(* Logix 5000 project; controller R5_CSS vendor 1 type 14 code 74 rev 19.11; software revision 19.01; part 4 of 20 *)
(* tags used below, declared in another part *)
   AlarmMaster : DINT;
   Coal_Tank_Heel_Inches : REAL;
   FC101 : FLOW_CONTROL;   // QUENCH BASIN FLOW TRANSMITTER CONTROL
   FC108 : FLOW_CONTROL;   // QUENCH FEED FLOW TRANSMITTER
   FC140A : FLOW_CONTROL;   // QUENCH TOWER UPPER SPRAY FLOW CONTROL
   FC140B : FLOW_CONTROL;   // QUENCH TOWER LOWER SPRAY FLOW CONTROL
   FC403 : FLOW_CONTROL;   // COALESCER FLOW CONTROLLER FEEDS TCV108
   FCV410_LT_Hold : BOOL;
   FlowControlForce : BOOL;
   FlowControlForceONS : BOOL;
   FT101_SCP : SCLP;   // QUENCH BASIN FLOW TRANSMITTER SCALER
   FT108_SCP : SCLP;   // QUENCH FEED FLOW TRANSMITTER SCALER
   FT140A_SCP : SCLP;   // QUENCH TOWER UPPER SPRAY FIT SCALER
   FT140ABFlowMeterFailed : BOOL;
   FT140B_SCP : SCLP;   // QUENCH TOWER LOWER SPRAY FLOW TRANSMITTER SCALER
   FT403_SCP : SCLP;   // QUENCH CONDITIONING QUENCH WATER PHASE FLOW SCALER
   LC101 : LEVEL_CONTROL;   // QUENCH TOWER BASIN LIT
   LC101_LT_Temp : REAL;
   LC304 : LEVEL_CONTROL;   // SETTLER SECONDARY TANK INTERFACE LEVEL
   LC304_LT_Raw : REAL;
   LevelControlForce : BOOL;
   LevelControlForceONS : BOOL;
   LossOfSignal_mA : DINT;
   LT101_SCP : SCLP;   // QUENCH TOWER BASIN LIT SCALER
   LT304_SCP : SCLP;   // QUENCH COALESCING SEPARATOR SECONDARY CHAMBER LEVEL SCALER
   PC132 : PRESSURE_CONTROL;
   PC132_SCP : SCLP;
   PC133 : PRESSURE_CONTROL;
   PC133_SCP : SCLP;
   PC134 : PRESSURE_CONTROL;
   PC134_SCP : SCLP;
   PC408 : PRESSURE_CONTROL;
   PDT408_SCP : SCLP;
   QuenchFlowAutoControl : BOOL;
   QuenchFlowAutoControlPB : BOOL;
   QuenchFlowAutoControlPB_ONS : BOOL;
   QuenchFlowMeterFailed : BOOL;
   QuenchFlowMeterFailedTOF : TIMER;
   TC101A : TEMP_CONTROL;   // QUENCH BASIN TRANSFER BASIN A TEMPERATURE CONTROL
   TC101B : TEMP_CONTROL;   // QUENCH BASIN TRANSFER BASIN B TEMPERATURE CONTROL
   TC110 : TEMP_CONTROL;   // Quench Water Cartridge Heater Bundle Temp
   TC110_SCP : SCLP;
   TC112 : TEMP_CONTROL;   // Quench Water Cartridge Heater ProcessTemp
   TC112_SCP : SCLP;
   TC114A : TEMP_CONTROL;   // QUENCH BASIN SHELL TEMPERATURE CONTROL
   TC114B : TEMP_CONTROL;   // QUENCH BASIN LIQUID TEMPERATURE CONTROL
   TC121C : TEMP_CONTROL;   // GTL FROM PRUC TEMPERATURE CONTROL
   TC121D : TEMP_CONTROL;   // GTL FROM PRUD TEMPERATURE CONTROL
   TC121E : TEMP_CONTROL;
   TC121F : TEMP_CONTROL;
   TC121G : TEMP_CONTROL;
   TC121H : TEMP_CONTROL;
   TC123A : TEMP_CONTROL;   // HEAT JACKET VENT FROM PRUA TEMPERATURE CONTROL
   TC123A_SCP : SCLP;   // HEAT JACKET VENT FROM PRUA TEMPERATURE TRANSMITTER SCALER
   TC123B : TEMP_CONTROL;
   TC123B_SCP : SCLP;   // HEAT JACKET VENT FROM PRUB TEMPERATURE TRANSMITTER SCALER
   TC123C : TEMP_CONTROL;   // HEAT JACKET VENT FROM PRUC TEMPERATURE CONTROL
   TC123C_SCP : SCLP;   // HEAT JACKET VENT FROM PRUC TEMPERATURE TRANSMITTER SCALER
   TC123D : TEMP_CONTROL;   // HEAT JACKET VENT FROM PRUD TEMPERATURE TRANSMITTER
   TC123D_SCP : SCLP;   // HEAT JACKET VENT FROM PRUD TEMPERATURE TRANSMITTER SCALER
   TC123E : TEMP_CONTROL;
   TC123E_SCP : SCLP;
   TC123F : TEMP_CONTROL;
   TC123F_SCP : SCLP;
   TC123G : TEMP_CONTROL;
   TC123G_SCP : SCLP;
   TC123H : TEMP_CONTROL;
   TC123H_SCP : SCLP;
   TC135 : TEMP_CONTROL;
   TC135_SCP : SCLP;
   TC136 : TEMP_CONTROL;
   TC136_SCP : SCLP;
   TC137 : TEMP_CONTROL;
   TC137_SCP : SCLP;
   TC215 : TEMP_CONTROL;   // OVERHEAD CONDENSER CHILLED WATER TEMPERATURE TRANSMITTER CONTROL
   TC215_SCP : SCLP;   // OVERHEAD CONDENSER CHILLED WATER TEMPERATURE TRANSMITTER SCALER
   TC216 : TEMP_CONTROL;   // OVERHEAD CONDENSER BASIN TEMPERATURE CONTROL
   TC217 : TEMP_CONTROL;   // OVERHEAD CONDENSED CHILLED WATER RETURN TEMPERATURE CONTROL
   TC218 : TEMP_CONTROL;   // OVERHEAD CONDENSER CHILLED WATER SUPPLY TEMPERATURE CONTROL
   TC313A : TEMP_CONTROL;   // PRIMARY COALESCER SEPARATOR TEMPERATURE CONTROL
   TC313B : TEMP_CONTROL;   // PRIMARY COALESCER SHELL TEMPERATURE CONTROL
   TC319 : TEMP_CONTROL;   // COALESCER OIL CHAMBER PROCESS TEMPERATURE CONTROL
   TC319A : TEMP_CONTROL;   // COALESCER OIL CHAMBER SHEATH TEMPERATURE
   TC320 : TEMP_CONTROL;   // COALESCER OIL CHAMBER SHELL TEMPERATURE TRANSMITTER CONTROL
   TC321A : TEMP_CONTROL;   // COALESCER OIL CHAMBER TRANSFER PUMP A TEMPERATURE TRANSMITTER
   TC321B : TEMP_CONTROL;   // COALESCER OIL CHAMBER TRANSFER PUMP B TEMPERATURE TRANSMITTER
   TC406 : TEMP_CONTROL;   // PROCESS WATER POST HX TEMPERATURE CONTROL
   TC406_SCP : SCLP;   // PROCESS WATER POST HX TEMPERATURE TRANSMITTER SCALER
   TC409 : TEMP_CONTROL;   // HX COOLING WATER SUPPLY TEMPERATURE CONTROL
   TC409_SCP : SCLP;   // HX COOLING WATER SUPPLY TEMPERATURE TRANSMITTER SCALER
   TC410 : TEMP_CONTROL;   // HX COOLING WATER RETURN TEMPERATURE CONTROL
   TC410_SCP : SCLP;   // HX COOLING WATER RETURN TEMPERATURE TRANSMITTER SCALER
   TT101A_SCP : SCLP;   // QUENCH BASIN TRANSFER BASIN A TEMPERATURE TRANSMITTER SCALER
   TT101B_SCP : SCLP;   // QUENCH BASIN TRANSFER BASIN B TEMPERATURE TRANSMITTER SCALER
   TT114A_SCP : SCLP;   // QUENCH BASIN SHELL TEMPERATURE TRANSMITTER SCALER
   TT114B_SCP : SCLP;   // QUENCH BASIN LIQUID TEMPERATURE TRANSMITTER SCALER
   TT121C_SCP : SCLP;
   TT121D_SCP : SCLP;
   TT121E_SCP : SCLP;
   TT121F_SCP : SCLP;   // GTL FROM PRUB TEMPERATURE TRANSMITTER SCALER
   TT121G_SCP : SCLP;   // GTL FROM PRUC TEMPERATURE TRANSMITTER SCALER
   TT121H_SCP : SCLP;   // GTL FROM PRUD TEMPERATURE TRANSMITTER SCALER
   TT216_SCP : SCLP;   // OVERHEAD CONDENSER BASIN TEMPERATURE TRANSMITTER SCALER
   TT217_SCP : SCLP;   // OVERHEAD CONDENSED CHILLED WATER RETURN TEMPERATURE TRANSMITTER
   TT218_SCP : SCLP;   // OVERHEAD CONDENSER CHILLED WATER SUPPLY TEMPERATURE SCALER
   TT313A_SCP : SCLP;   // PRIMARY COALESCER SEPARATOR TEMPERATURE TRANSMITTER SCALER
   TT313B_SCP : SCLP;   // PRIMARY COALESCER SHELL TEMPERATURE TRANSMITTER SCALER
   TT319_SCP : SCLP;   // COALESCER OIL CHAMBER SHELL TEMPERATURE TRANSMITTER SCALER
   TT319A_SCP : SCLP;
   TT320_SCP : SCLP;   // COALESCER OIL CHAMBER SHELL TEMPERATURE TRANSMITTER SCALER
   TT321A_SCP : SCLP;   // COALESCER OIL CHAMBER TRANSFER PUMP A TEMPERATURE TRANSMITTER SCALER
   TT321B_SCP : SCLP;   // COALESCER OIL CHAMBER TRANSFER PUMP B TEMPERATURE TRANSMITTER
(* MainProgram, continued *)

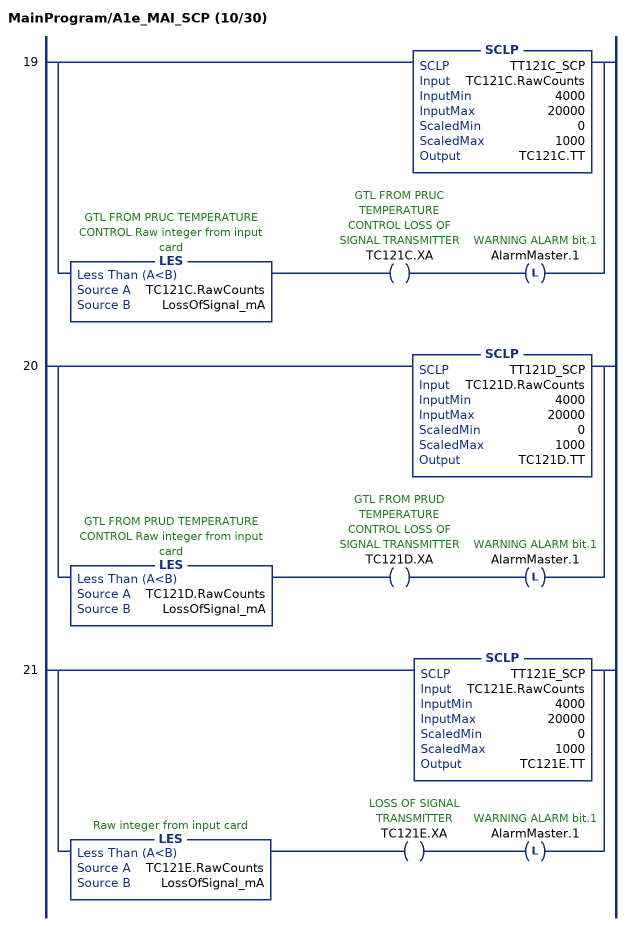
   [picture p54: MainProgram/A1e_MAI_SCP rungs 19-21]
   19: [SCLP(TT121C_SCP,TC121C.RawCounts,4000,20000,0,1000,TC121C.TT) ,LES(TC121C.RawCounts,LossOfSignal_mA) OTE(TC121C.XA) OTL(AlarmMaster.1) ];
   20: [SCLP(TT121D_SCP,TC121D.RawCounts,4000,20000,0,1000,TC121D.TT) ,LES(TC121D.RawCounts,LossOfSignal_mA) OTE(TC121D.XA) OTL(AlarmMaster.1) ];
   21: [SCLP(TT121E_SCP,TC121E.RawCounts,4000,20000,0,1000,TC121E.TT) ,LES(TC121E.RawCounts,LossOfSignal_mA) OTE(TC121E.XA) OTL(AlarmMaster.1) ];
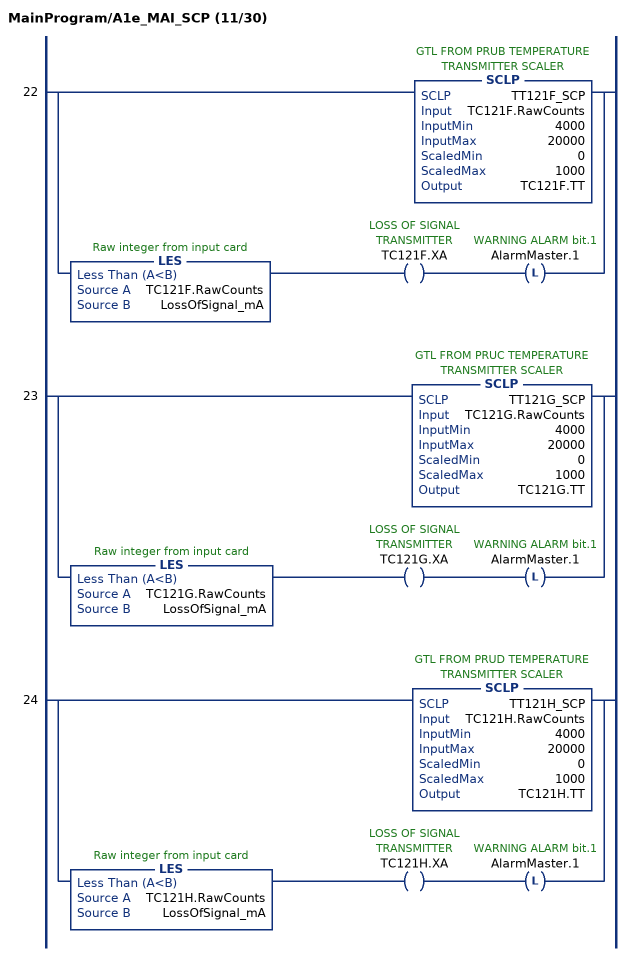
   22: [SCLP(TT121F_SCP,TC121F.RawCounts,4000,20000,0,1000,TC121F.TT) ,LES(TC121F.RawCounts,LossOfSignal_mA) OTE(TC121F.XA) OTL(AlarmMaster.1) ];
   23: [SCLP(TT121G_SCP,TC121G.RawCounts,4000,20000,0,1000,TC121G.TT) ,LES(TC121G.RawCounts,LossOfSignal_mA) OTE(TC121G.XA) OTL(AlarmMaster.1) ];
   24: [SCLP(TT121H_SCP,TC121H.RawCounts,4000,20000,0,1000,TC121H.TT) ,LES(TC121H.RawCounts,LossOfSignal_mA) OTE(TC121H.XA) OTL(AlarmMaster.1) ];
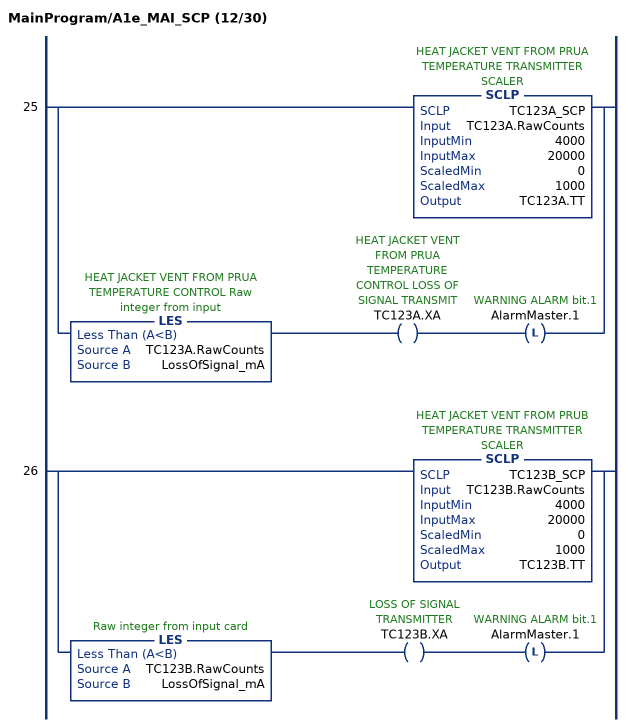
   25: [SCLP(TC123A_SCP,TC123A.RawCounts,4000,20000,0,1000,TC123A.TT) ,LES(TC123A.RawCounts,LossOfSignal_mA) OTE(TC123A.XA) OTL(AlarmMaster.1) ];
   26: [SCLP(TC123B_SCP,TC123B.RawCounts,4000,20000,0,1000,TC123B.TT) ,LES(TC123B.RawCounts,LossOfSignal_mA) OTE(TC123B.XA) OTL(AlarmMaster.1) ];
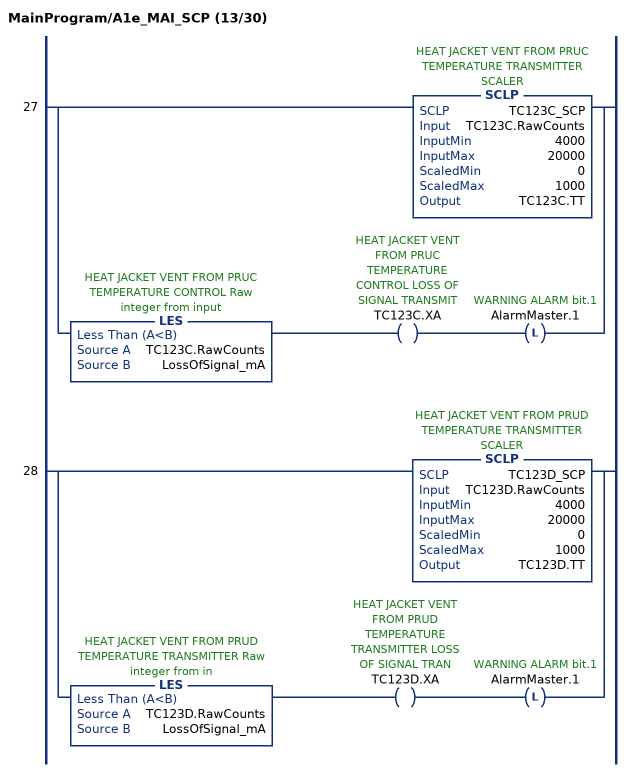
   27: [SCLP(TC123C_SCP,TC123C.RawCounts,4000,20000,0,1000,TC123C.TT) ,LES(TC123C.RawCounts,LossOfSignal_mA) OTE(TC123C.XA) OTL(AlarmMaster.1) ];
   28: [SCLP(TC123D_SCP,TC123D.RawCounts,4000,20000,0,1000,TC123D.TT) ,LES(TC123D.RawCounts,LossOfSignal_mA) OTE(TC123D.XA) OTL(AlarmMaster.1) ];
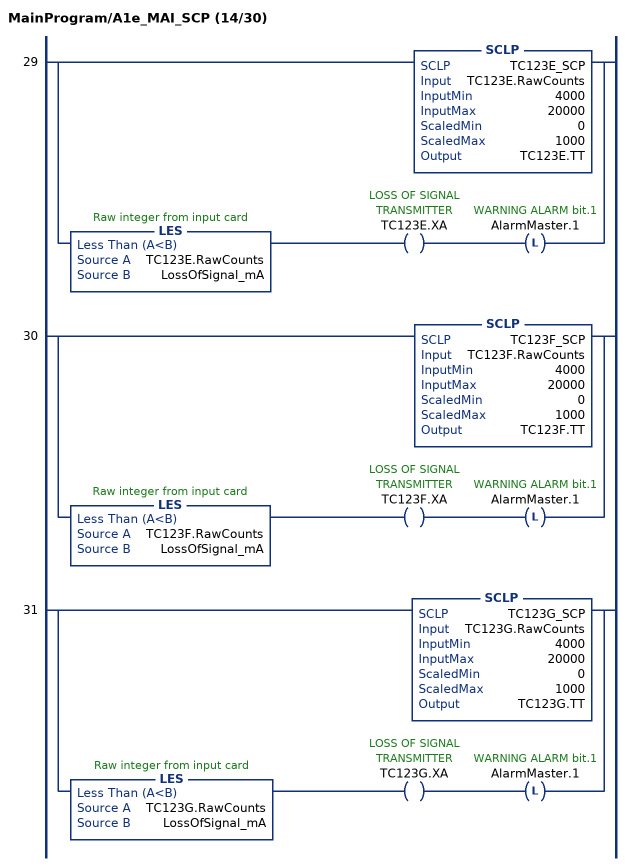
   29: [SCLP(TC123E_SCP,TC123E.RawCounts,4000,20000,0,1000,TC123E.TT) ,LES(TC123E.RawCounts,LossOfSignal_mA) OTE(TC123E.XA) OTL(AlarmMaster.1) ];
   30: [SCLP(TC123F_SCP,TC123F.RawCounts,4000,20000,0,1000,TC123F.TT) ,LES(TC123F.RawCounts,LossOfSignal_mA) OTE(TC123F.XA) OTL(AlarmMaster.1) ];
   31: [SCLP(TC123G_SCP,TC123G.RawCounts,4000,20000,0,1000,TC123G.TT) ,LES(TC123G.RawCounts,LossOfSignal_mA) OTE(TC123G.XA) OTL(AlarmMaster.1) ];
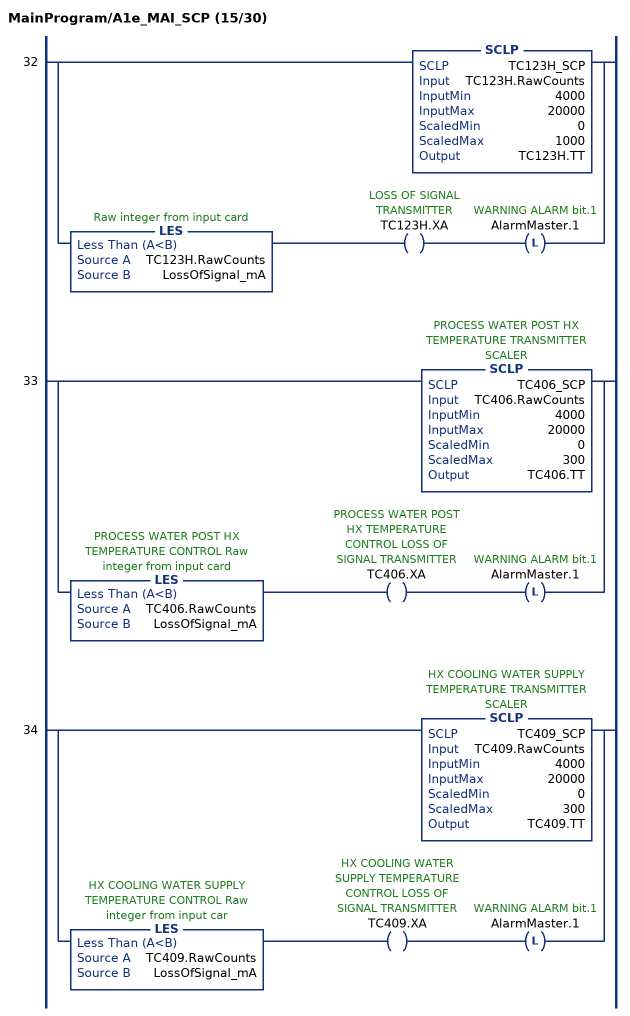
   32: [SCLP(TC123H_SCP,TC123H.RawCounts,4000,20000,0,1000,TC123H.TT) ,LES(TC123H.RawCounts,LossOfSignal_mA) OTE(TC123H.XA) OTL(AlarmMaster.1) ];
   33: [SCLP(TC406_SCP,TC406.RawCounts,4000,20000,0,300,TC406.TT) ,LES(TC406.RawCounts,LossOfSignal_mA) OTE(TC406.XA) OTL(AlarmMaster.1) ];
   34: [SCLP(TC409_SCP,TC409.RawCounts,4000,20000,0,300,TC409.TT) ,LES(TC409.RawCounts,LossOfSignal_mA) OTE(TC409.XA) OTL(AlarmMaster.1) ];
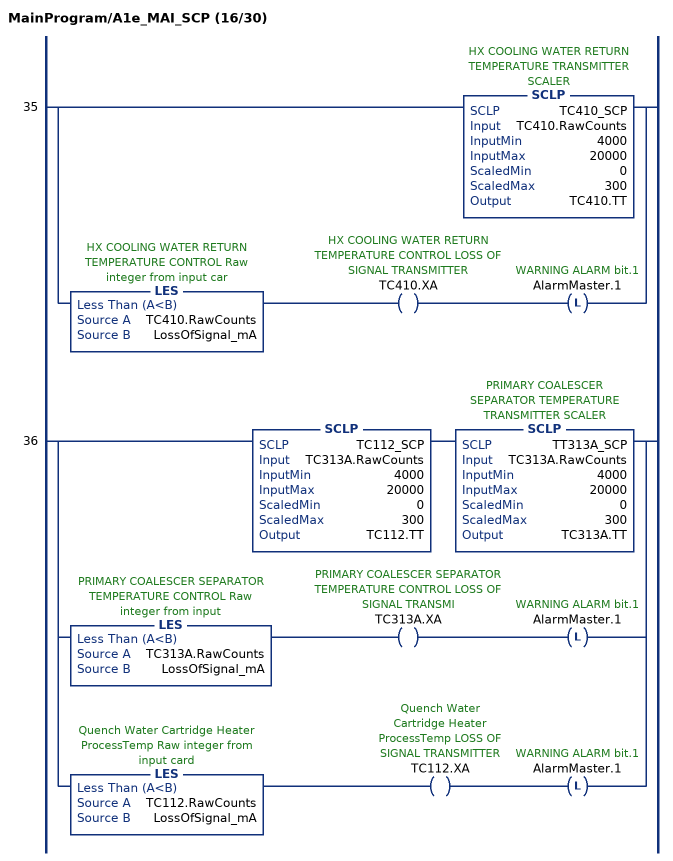
   35: [SCLP(TC410_SCP,TC410.RawCounts,4000,20000,0,300,TC410.TT) ,LES(TC410.RawCounts,LossOfSignal_mA) OTE(TC410.XA) OTL(AlarmMaster.1) ];
   36: [SCLP(TC112_SCP,TC313A.RawCounts,4000,20000,0,300,TC112.TT) SCLP(TT313A_SCP,TC313A.RawCounts,4000,20000,0,300,TC313A.TT) ,LES(TC313A.RawCounts,LossOfSignal_mA) OTE(TC313A.XA) OTL(AlarmMaster.1) ,LES(TC112.RawCounts,LossOfSignal_mA) OTE(TC112.XA) OTL(AlarmMaster.1) ];
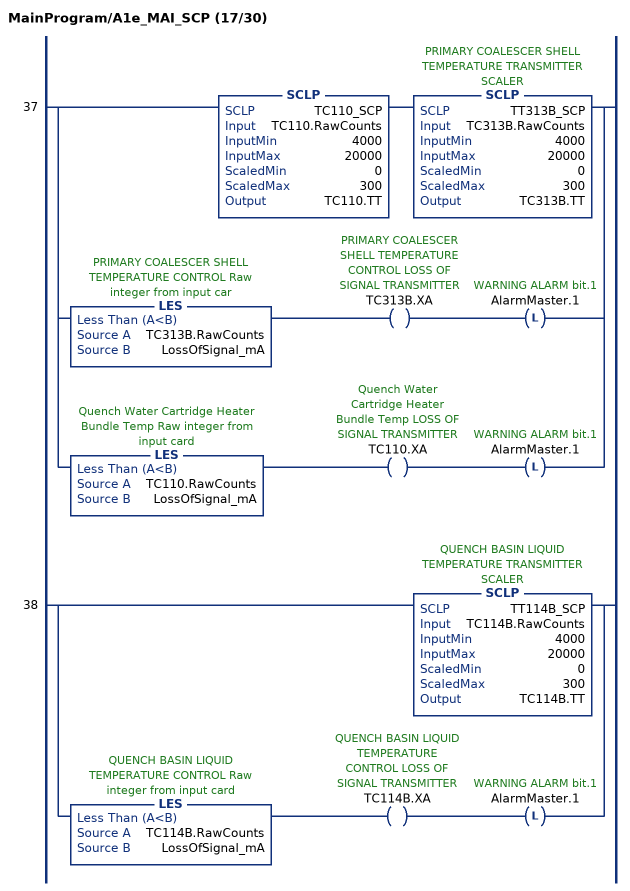
   37: [SCLP(TC110_SCP,TC110.RawCounts,4000,20000,0,300,TC110.TT) SCLP(TT313B_SCP,TC313B.RawCounts,4000,20000,0,300,TC313B.TT) ,LES(TC313B.RawCounts,LossOfSignal_mA) OTE(TC313B.XA) OTL(AlarmMaster.1) ,LES(TC110.RawCounts,LossOfSignal_mA) OTE(TC110.XA) OTL(AlarmMaster.1) ];
   38: [SCLP(TT114B_SCP,TC114B.RawCounts,4000,20000,0,300,TC114B.TT) ,LES(TC114B.RawCounts,LossOfSignal_mA) OTE(TC114B.XA) OTL(AlarmMaster.1) ];
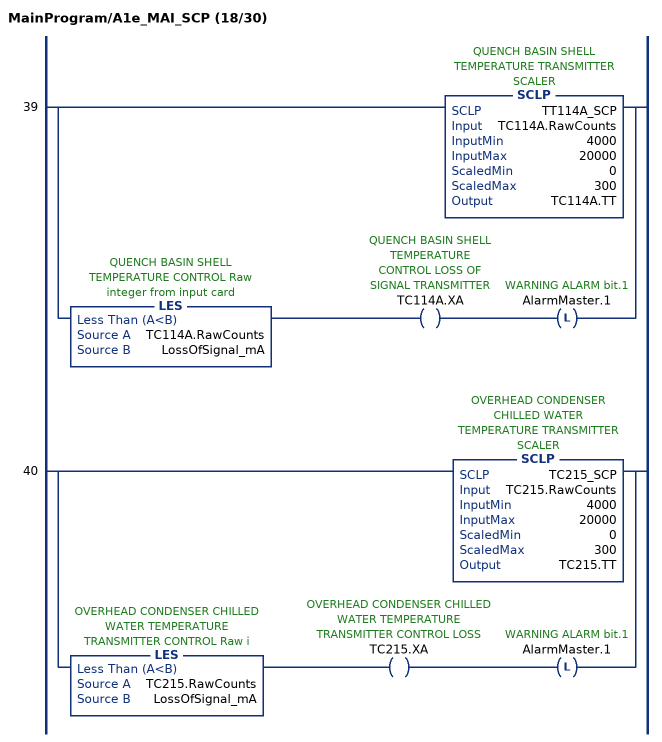
   39: [SCLP(TT114A_SCP,TC114A.RawCounts,4000,20000,0,300,TC114A.TT) ,LES(TC114A.RawCounts,LossOfSignal_mA) OTE(TC114A.XA) OTL(AlarmMaster.1) ];
   40: [SCLP(TC215_SCP,TC215.RawCounts,4000,20000,0,300,TC215.TT) ,LES(TC215.RawCounts,LossOfSignal_mA) OTE(TC215.XA) OTL(AlarmMaster.1) ];
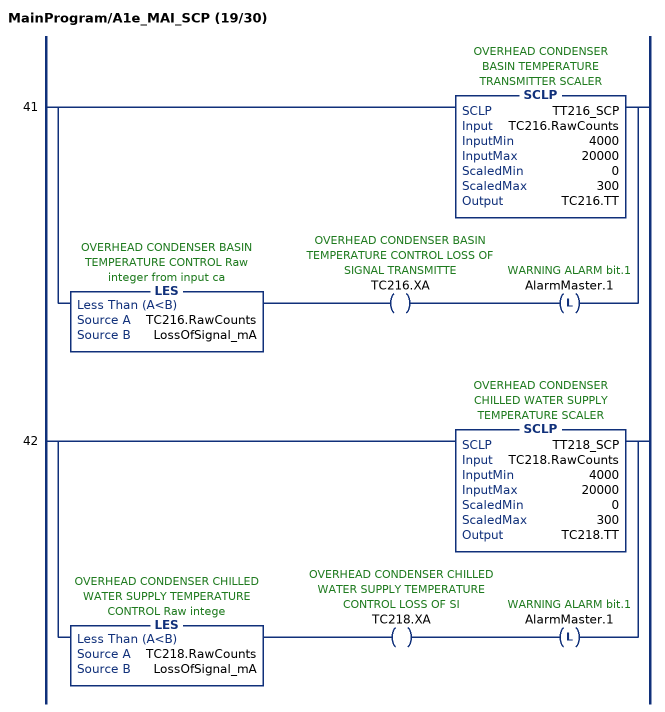
   41: [SCLP(TT216_SCP,TC216.RawCounts,4000,20000,0,300,TC216.TT) ,LES(TC216.RawCounts,LossOfSignal_mA) OTE(TC216.XA) OTL(AlarmMaster.1) ];
   42: [SCLP(TT218_SCP,TC218.RawCounts,4000,20000,0,300,TC218.TT) ,LES(TC218.RawCounts,LossOfSignal_mA) OTE(TC218.XA) OTL(AlarmMaster.1) ];
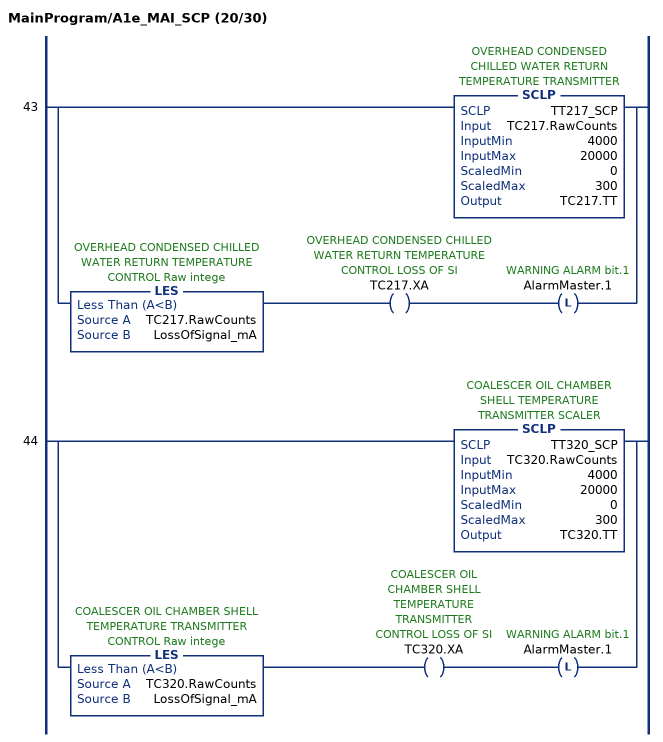
   43: [SCLP(TT217_SCP,TC217.RawCounts,4000,20000,0,300,TC217.TT) ,LES(TC217.RawCounts,LossOfSignal_mA) OTE(TC217.XA) OTL(AlarmMaster.1) ];
   44: [SCLP(TT320_SCP,TC320.RawCounts,4000,20000,0,300,TC320.TT) ,LES(TC320.RawCounts,LossOfSignal_mA) OTE(TC320.XA) OTL(AlarmMaster.1) ];
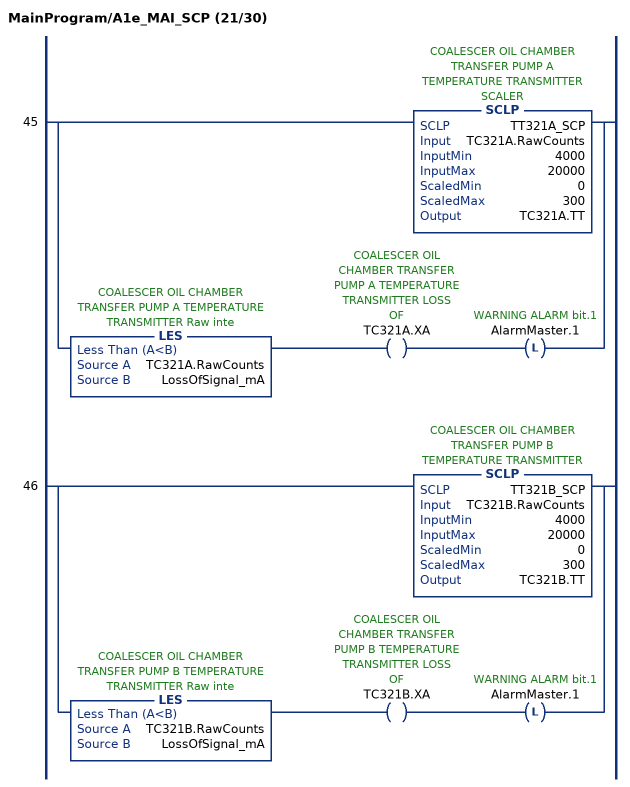
   45: [SCLP(TT321A_SCP,TC321A.RawCounts,4000,20000,0,300,TC321A.TT) ,LES(TC321A.RawCounts,LossOfSignal_mA) OTE(TC321A.XA) OTL(AlarmMaster.1) ];
   46: [SCLP(TT321B_SCP,TC321B.RawCounts,4000,20000,0,300,TC321B.TT) ,LES(TC321B.RawCounts,LossOfSignal_mA) OTE(TC321B.XA) OTL(AlarmMaster.1) ];
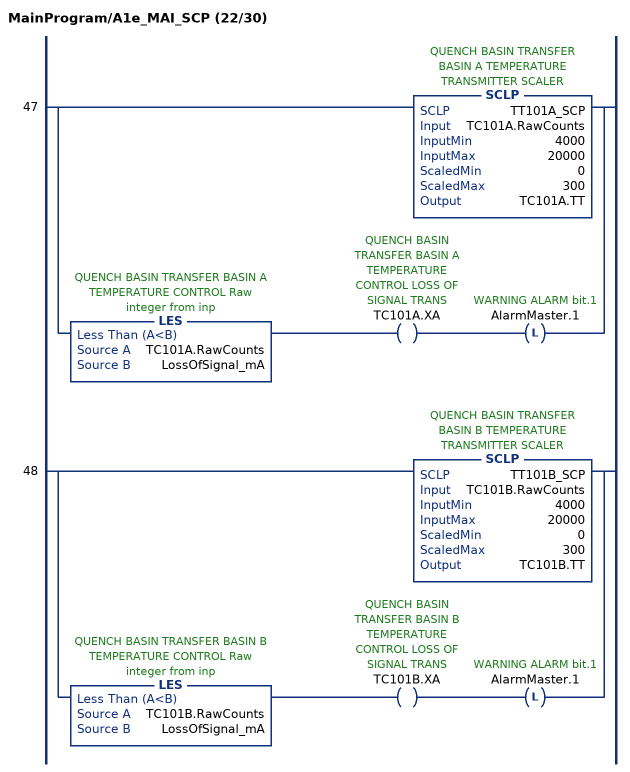
   47: [SCLP(TT101A_SCP,TC101A.RawCounts,4000,20000,0,300,TC101A.TT) ,LES(TC101A.RawCounts,LossOfSignal_mA) OTE(TC101A.XA) OTL(AlarmMaster.1) ];
   48: [SCLP(TT101B_SCP,TC101B.RawCounts,4000,20000,0,300,TC101B.TT) ,LES(TC101B.RawCounts,LossOfSignal_mA) OTE(TC101B.XA) OTL(AlarmMaster.1) ];
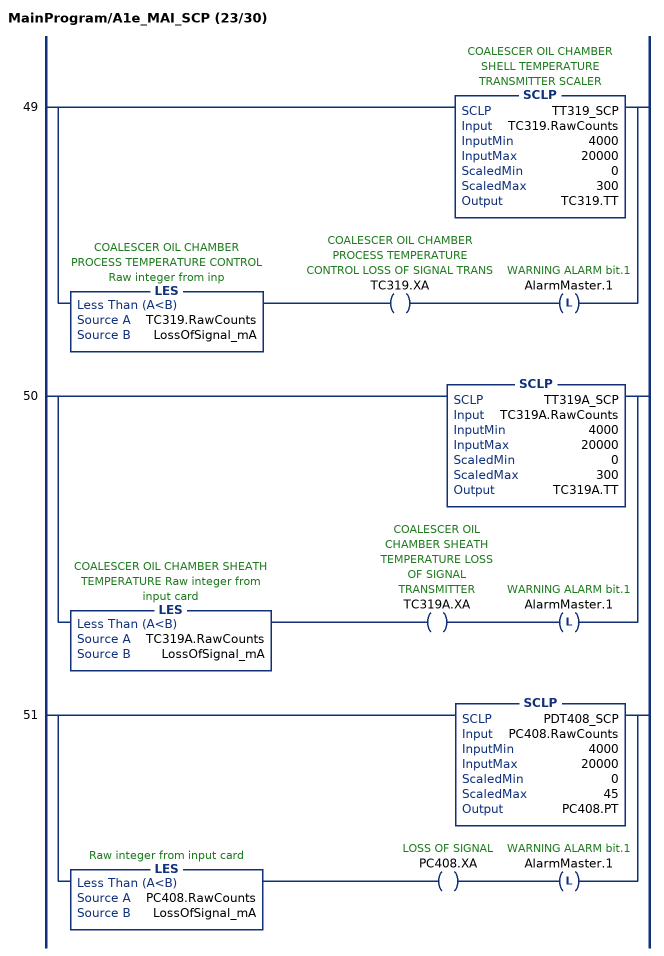
   49: [SCLP(TT319_SCP,TC319.RawCounts,4000,20000,0,300,TC319.TT) ,LES(TC319.RawCounts,LossOfSignal_mA) OTE(TC319.XA) OTL(AlarmMaster.1) ];
   50: [SCLP(TT319A_SCP,TC319A.RawCounts,4000,20000,0,300,TC319A.TT) ,LES(TC319A.RawCounts,LossOfSignal_mA) OTE(TC319A.XA) OTL(AlarmMaster.1) ];
   51: [SCLP(PDT408_SCP,PC408.RawCounts,4000,20000,0,45,PC408.PT) ,LES(PC408.RawCounts,LossOfSignal_mA) OTE(PC408.XA) OTL(AlarmMaster.1) ];
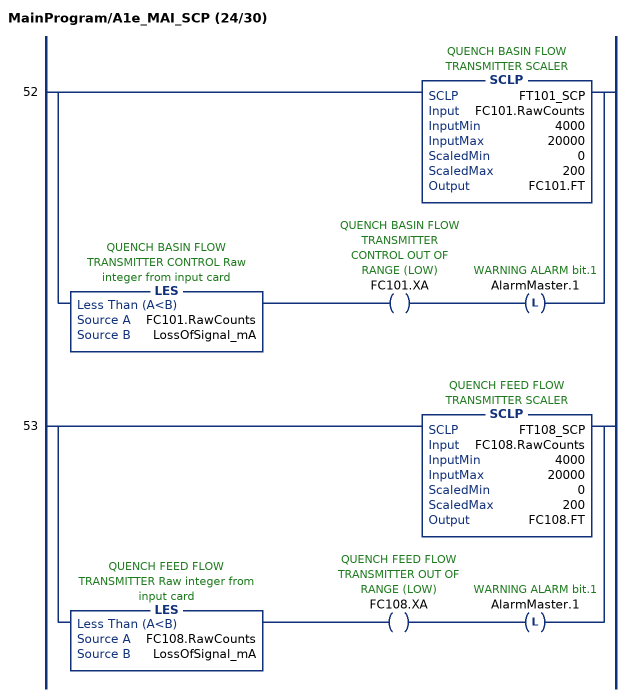
   52: [SCLP(FT101_SCP,FC101.RawCounts,4000,20000,0,200,FC101.FT) ,LES(FC101.RawCounts,LossOfSignal_mA) OTE(FC101.XA) OTL(AlarmMaster.1) ];
   53: [SCLP(FT108_SCP,FC108.RawCounts,4000,20000,0,200,FC108.FT) ,LES(FC108.RawCounts,LossOfSignal_mA) OTE(FC108.XA) OTL(AlarmMaster.1) ];
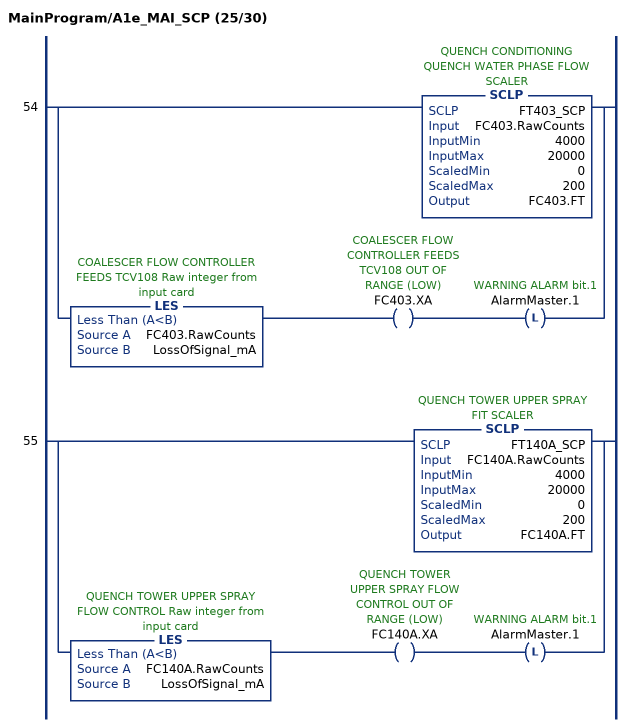
   54: [SCLP(FT403_SCP,FC403.RawCounts,4000,20000,0,200,FC403.FT) ,LES(FC403.RawCounts,LossOfSignal_mA) OTE(FC403.XA) OTL(AlarmMaster.1) ];
   55: [SCLP(FT140A_SCP,FC140A.RawCounts,4000,20000,0,200,FC140A.FT) ,LES(FC140A.RawCounts,LossOfSignal_mA) OTE(FC140A.XA) OTL(AlarmMaster.1) ];
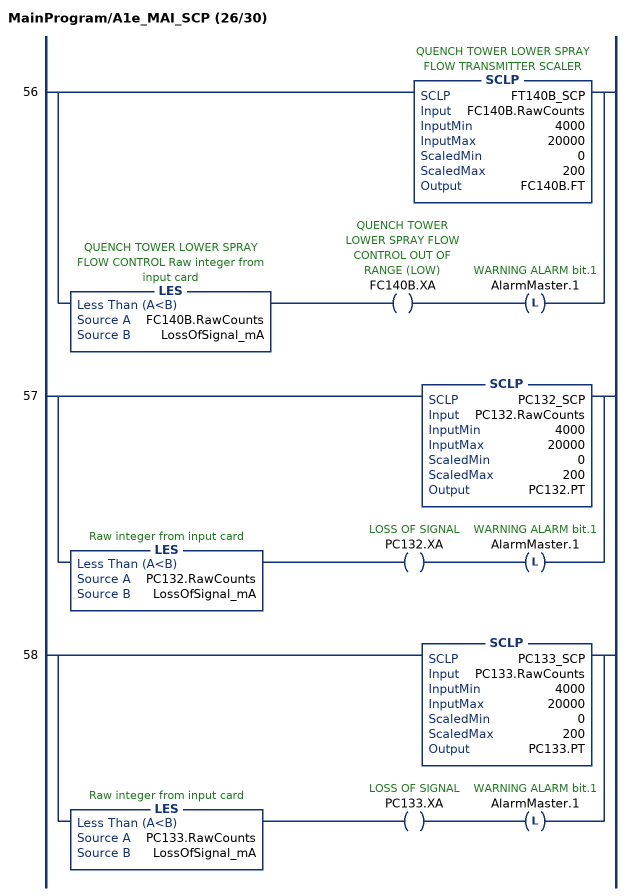
   56: [SCLP(FT140B_SCP,FC140B.RawCounts,4000,20000,0,200,FC140B.FT) ,LES(FC140B.RawCounts,LossOfSignal_mA) OTE(FC140B.XA) OTL(AlarmMaster.1) ];
   57: [SCLP(PC132_SCP,PC132.RawCounts,4000,20000,0,200,PC132.PT) ,LES(PC132.RawCounts,LossOfSignal_mA) OTE(PC132.XA) OTL(AlarmMaster.1) ];
   58: [SCLP(PC133_SCP,PC133.RawCounts,4000,20000,0,200,PC133.PT) ,LES(PC133.RawCounts,LossOfSignal_mA) OTE(PC133.XA) OTL(AlarmMaster.1) ];
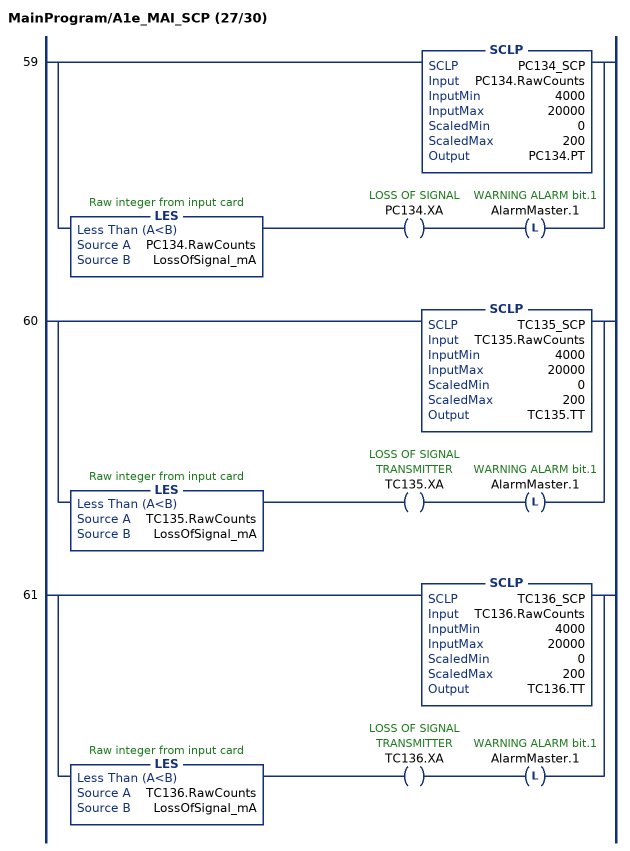
   59: [SCLP(PC134_SCP,PC134.RawCounts,4000,20000,0,200,PC134.PT) ,LES(PC134.RawCounts,LossOfSignal_mA) OTE(PC134.XA) OTL(AlarmMaster.1) ];
   60: [SCLP(TC135_SCP,TC135.RawCounts,4000,20000,0,200,TC135.TT) ,LES(TC135.RawCounts,LossOfSignal_mA) OTE(TC135.XA) OTL(AlarmMaster.1) ];
   61: [SCLP(TC136_SCP,TC136.RawCounts,4000,20000,0,200,TC136.TT) ,LES(TC136.RawCounts,LossOfSignal_mA) OTE(TC136.XA) OTL(AlarmMaster.1) ];
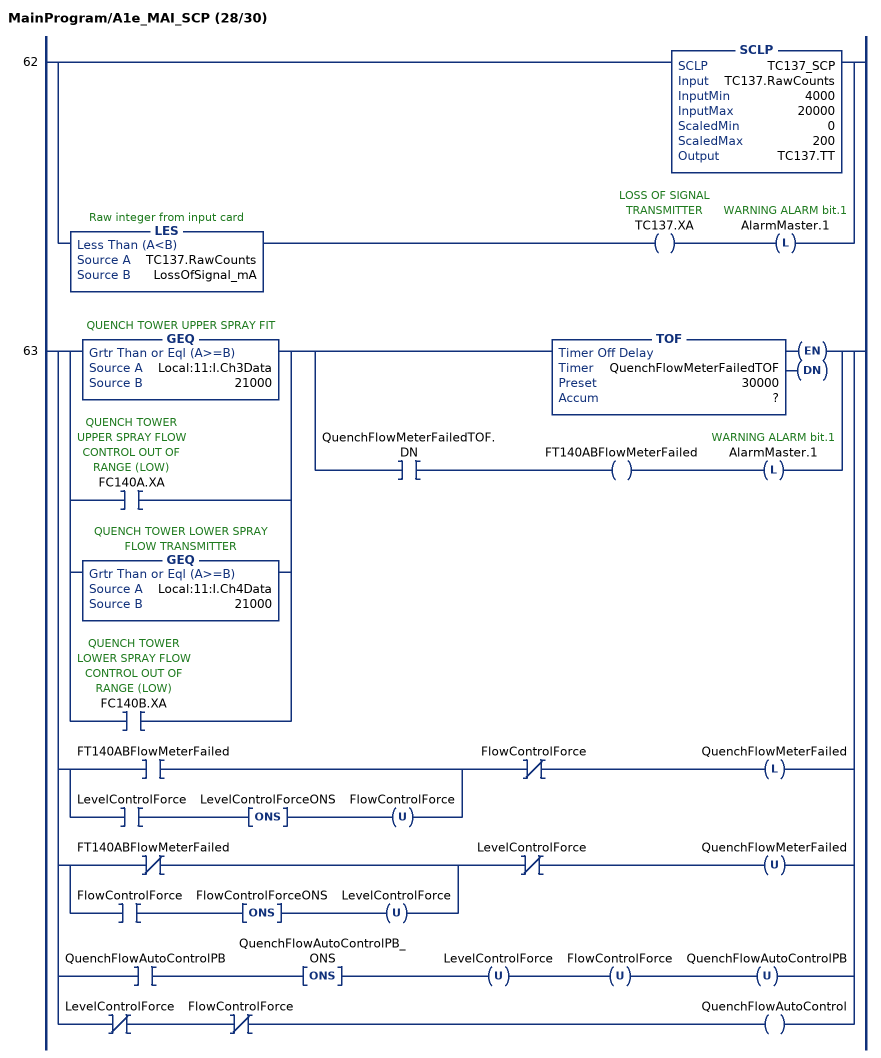
   62: [SCLP(TC137_SCP,TC137.RawCounts,4000,20000,0,200,TC137.TT) ,LES(TC137.RawCounts,LossOfSignal_mA) OTE(TC137.XA) OTL(AlarmMaster.1) ];
   63: [[GEQ(Local:11:I.Ch3Data,21000) ,XIC(FC140A.XA) ,GEQ(Local:11:I.Ch4Data,21000) ,XIC(FC140B.XA) ] [TOF(QuenchFlowMeterFailedTOF,?,?) ,XIC(QuenchFlowMeterFailedTOF.DN) OTE(FT140ABFlowMeterFailed) OTL(AlarmMaster.1) ] ,[XIC(FT140ABFlowMeterFailed) ,XIC(LevelControlForce) ONS(LevelControlForceONS) OTU(FlowControlForce) ] XIO(FlowControlForce) OTL(QuenchFlowMeterFailed) ,[XIO(FT140ABFlowMeterFailed) ,XIC(FlowControlForce) ONS(FlowControlForceONS) OTU(LevelControlForce) ] XIO(LevelControlForce) OTU(QuenchFlowMeterFailed) ,XIC(QuenchFlowAutoControlPB) ONS(QuenchFlowAutoControlPB_ONS) OTU(LevelControlForce) OTU(FlowControlForce) OTU(QuenchFlowAutoControlPB) ,XIO(LevelControlForce) XIO(FlowControlForce) OTE(QuenchFlowAutoControl) ];
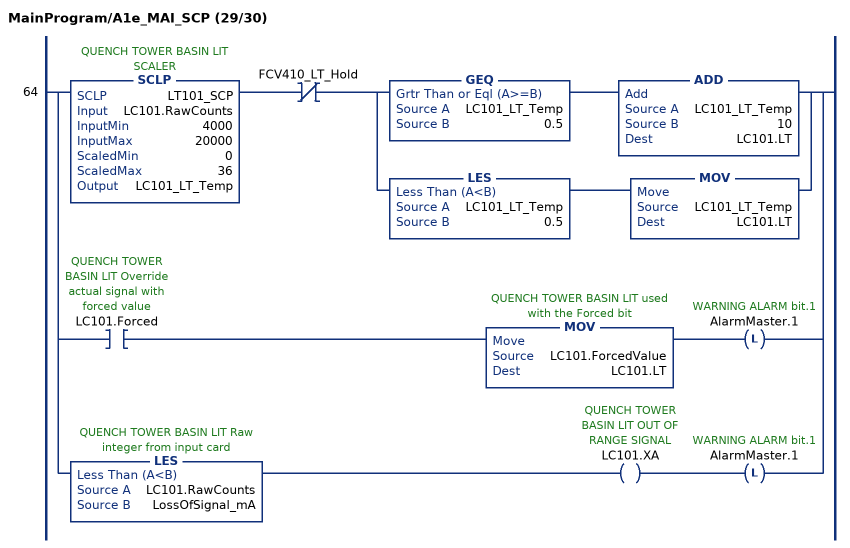
   64: [SCLP(LT101_SCP,LC101.RawCounts,4000,20000,0,36,LC101_LT_Temp) XIO(FCV410_LT_Hold) [GEQ(LC101_LT_Temp,0.5) ADD(LC101_LT_Temp,10,LC101.LT) ,LES(LC101_LT_Temp,0.5) MOV(LC101_LT_Temp,LC101.LT) ] ,XIC(LC101.Forced) MOV(LC101.ForcedValue,LC101.LT) OTL(AlarmMaster.1) ,LES(LC101.RawCounts,LossOfSignal_mA) OTE(LC101.XA) OTL(AlarmMaster.1) ];
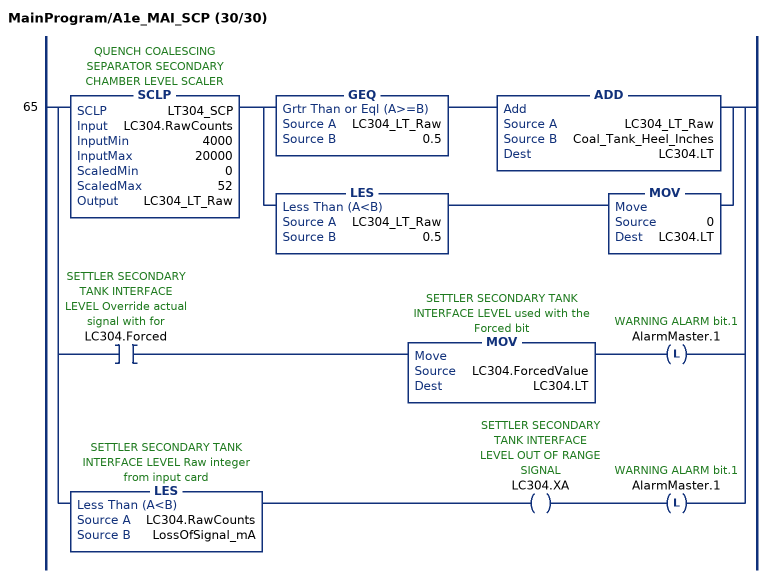
   65: [SCLP(LT304_SCP,LC304.RawCounts,4000,20000,0,52,LC304_LT_Raw) [GEQ(LC304_LT_Raw,0.5) ADD(LC304_LT_Raw,Coal_Tank_Heel_Inches,LC304.LT) ,LES(LC304_LT_Raw,0.5) MOV(0,LC304.LT) ] ,XIC(LC304.Forced) MOV(LC304.ForcedValue,LC304.LT) OTL(AlarmMaster.1) ,LES(LC304.RawCounts,LossOfSignal_mA) OTE(LC304.XA) OTL(AlarmMaster.1) ];
END_ROUTINE
